{attribute 'GeneratedUsingTerminal: EP2316-0008-0017'}
{attribute addProperty BoxType "EP2316-0008-0017"}
{attribute addProperty Id "DO_Diag_InputsAT %I*DO_Diag_Inputs_CC4551489DO_Diag_Inputs_1AT %I*DO_Diag_Inputs_212B82C19DO_Inputs_DeviceAT %I*DO_Inputs_Device_AF161A9E4DO_OutputsAT %Q*DO_Outputs_28AC1A9E8DO_Outputs_DeviceAT %Q*DO_Outputs_Device_36A5EF172WcStateAT %I*WcState_9091E0EB2InfoDataAT %I*InfoData_94A18F5E2"}
{attribute addProperty CRC "1468923339"}
{attribute addProperty Size "36"}
TYPE EP2316_578DFDCB EXTENDS EtcSlaveTerminalBase_947E5A46 :
STRUCT
	{attribute addProperty Name "DO_Diag_Inputs"}
	DO_Diag_Inputs : DO_Diag_Inputs_CC455148;
	{attribute addProperty Name "DO_Diag_Inputs_1"}
	DO_Diag_Inputs_1 : DO_Diag_Inputs_212B82C1;
	{attribute addProperty Name "DO_Inputs_Device"}
	DO_Inputs_Device : DO_Inputs_Device_AF161A9E;
	{attribute addProperty Name "DO_Outputs"}
	DO_Outputs : DO_Outputs_28AC1A9E;
	{attribute addProperty Name "DO_Outputs_Device"}
	DO_Outputs_Device : DO_Outputs_Device_36A5EF17;
	{attribute addProperty Name "WcState"}
	WcState : WcState_9091E0EB;
	{attribute addProperty Name "InfoData"}
	InfoData : InfoData_94A18F5E;
END_STRUCT
END_TYPE

(* stored: Version 1.2.0.0, ProductVersion 3.1.4024.9
   DUT EP2316_578DFDCB: Id {d82a26c4-ec74-4188-b0c0-a226cc3b6124} *)
